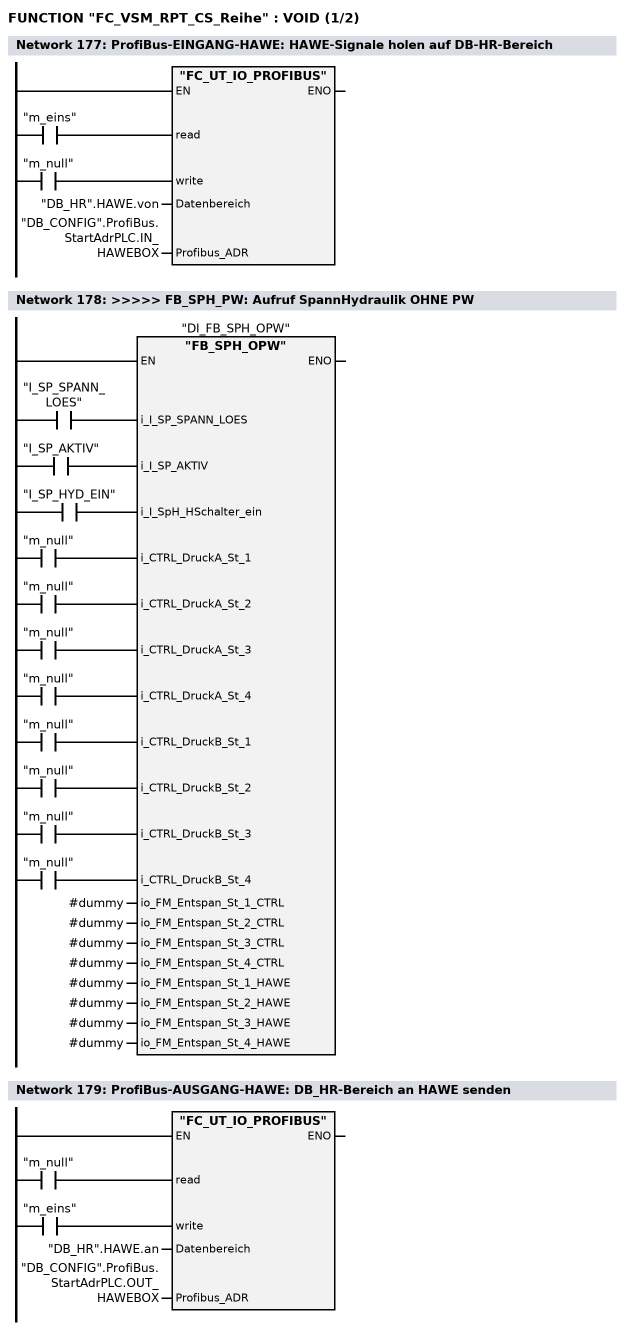

      U     "m_eins";
      =     L     21.0;
      BLD   103;
      U     "m_null";
      =     L     21.1;
      BLD   103;
      CALL "FC_UT_IO_PROFIBUS" (
           read                     := L     21.0,
           write                    := L     21.1,
           Datenbereich             := "DB_HR".HAWE.von,
           Profibus_ADR             := "DB_CONFIG".ProfiBus.StartAdrPLC.IN_HAWEBOX);
      NOP   0;
NETWORK
TITLE =>>>>> FB_SPH_PW: Aufruf SpannHydraulik OHNE PW

      U     "I_SP_SPANN_LOES";
      =     L     21.0;
      BLD   103;
      U     "I_SP_AKTIV";
      =     L     21.1;
      BLD   103;
      U     "I_SP_HYD_EIN";
      =     L     21.2;
      BLD   103;
      U     "m_null";
      =     L     21.3;
      BLD   103;
      U     "m_null";
      =     L     21.4;
      BLD   103;
      U     "m_null";
      =     L     21.5;
      BLD   103;
      U     "m_null";
      =     L     21.6;
      BLD   103;
      U     "m_null";
      =     L     21.7;
      BLD   103;
      U     "m_null";
      =     L     22.0;
      BLD   103;
      U     "m_null";
      =     L     22.1;
      BLD   103;
      U     "m_null";
      =     L     22.2;
      BLD   103;
      CALL "FB_SPH_OPW" , "DI_FB_SPH_OPW" (
           i_I_SP_SPANN_LOES        := L     21.0,
           i_I_SP_AKTIV             := L     21.1,
           i_I_SpH_HSchalter_ein    := L     21.2,
           i_CTRL_DruckA_St_1       := L     21.3,
           i_CTRL_DruckA_St_2       := L     21.4,
           i_CTRL_DruckA_St_3       := L     21.5,
           i_CTRL_DruckA_St_4       := L     21.6,
           i_CTRL_DruckB_St_1       := L     21.7,
           i_CTRL_DruckB_St_2       := L     22.0,
           i_CTRL_DruckB_St_3       := L     22.1,
           i_CTRL_DruckB_St_4       := L     22.2,
           io_FM_Entspan_St_1_CTRL  := #dummy,
           io_FM_Entspan_St_2_CTRL  := #dummy,
           io_FM_Entspan_St_3_CTRL  := #dummy,
           io_FM_Entspan_St_4_CTRL  := #dummy,
           io_FM_Entspan_St_1_HAWE  := #dummy,
           io_FM_Entspan_St_2_HAWE  := #dummy,
           io_FM_Entspan_St_3_HAWE  := #dummy,
           io_FM_Entspan_St_4_HAWE  := #dummy);
      NOP   0;
NETWORK
TITLE =ProfiBus-AUSGANG-HAWE: DB_HR-Bereich an HAWE senden

      U     "m_null";
      =     L     21.0;
      BLD   103;
      U     "m_eins";
      =     L     21.1;
      BLD   103;
      CALL "FC_UT_IO_PROFIBUS" (
           read                     := L     21.0,
           write                    := L     21.1,
           Datenbereich             := "DB_HR".HAWE.an,
           Profibus_ADR             := "DB_CONFIG".ProfiBus.StartAdrPLC.OUT_HAWEBOX);
      NOP   0;
NETWORK
TITLE =M-Ausgang: SpannHydraulik Pumpe ein
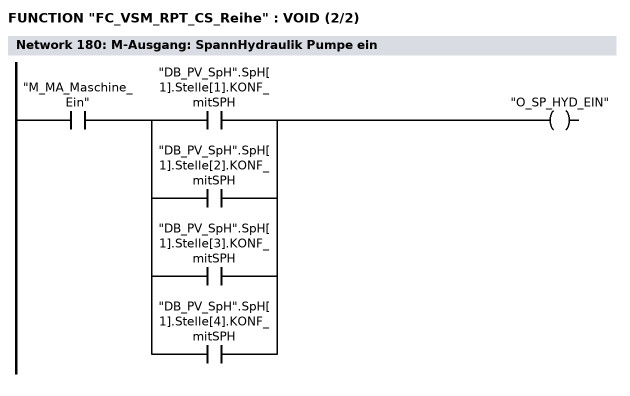

      U     "M_MA_Maschine_Ein";
      U(    ;
      O     "DB_PV_SpH".SpH[1].Stelle[1].KONF_mitSPH;
      O     "DB_PV_SpH".SpH[1].Stelle[2].KONF_mitSPH;
      O     "DB_PV_SpH".SpH[1].Stelle[3].KONF_mitSPH;
      O     "DB_PV_SpH".SpH[1].Stelle[4].KONF_mitSPH;
      )     ;
      =     "O_SP_HYD_EIN";
NETWORK
TITLE =Aufruf: Rüstplatztüre entriegeln

RPT:  CALL "FC_RPT_ENTRIEGELN" ;
      NOP   0;
END_FUNCTION

